PROGRAM TEST
VAR
	fbTest : FB_Test;
	
	i : INT;
END_VAR

i := fbTest.Prop;

END_PROGRAM

(* stored: Version 1.1.0.1, ProductVersion 3.1.4024.12
   POU TEST: Id {6cabfc6a-b673-4936-9b06-43f4016d3a05}, SpecialFunc None *)
